PROGRAM P4_01_Write
VAR
	stDBParam 				:ST_AuditTrail;	
	tableColumns			:ARRAY [0..5] OF STRING(50) := ['DateTime', 'User', 'Event', 'Description', 'OldValue', 'NewValue'];	

	fbDBWrite				:FB_PLCDBWriteEvt(sNetId:=CONST.AMS_NETID, tTimeout:=DEFAULT_ADS_TIMEOUT);	
	bWrite					:BOOL;
	

	
	fbRecipeProdValue		:ARRAY[0..9] OF FB_WriteChange;
	fbRecipeProdStrings		:ARRAY[0..9] OF FB_WriteChange_STR;
	fbRecipeProdClick		:ARRAY[0..9] OF FB_WriteClick;
	bRecipeProdChange		:ARRAY[0..19] OF BOOL;
	
	fbRecipeCleanValue		:ARRAY[0..29] OF FB_WriteChange;
	fbRecipeCleanStrings	:ARRAY[0..29] OF FB_WriteChange_STR;
	fbRecipeCleanClick		:ARRAY[0..29] OF FB_WriteClick;
	bRecipeCleanChange		:ARRAY[0..39] OF BOOL;
	
	fbBatchProdValue		:ARRAY[0..9] OF FB_WriteChange;
	fbBatchProdStrings		:ARRAY[0..9] OF FB_WriteChange_STR;
	fbBatchProdClick		:ARRAY[0..9] OF FB_WriteClick;
	bBatchProdChange		:ARRAY[0..19] OF BOOL;
	
	fbBatchCleanValue		:ARRAY[0..29] OF FB_WriteChange;
	fbBatchCleanStrings		:ARRAY[0..29] OF FB_WriteChange_STR;
	fbBatchCleanClick		:ARRAY[0..29] OF FB_WriteClick;
	bBatchCleanChange		:ARRAY[0..39] OF BOOL;
	
	
	fbSettingsChange		:ARRAY[0..19] OF FB_WriteChange;
	bSettingsChange			:ARRAY[0..19] OF BOOL;	
	
	fbAlarmsettChange		:ARRAY[0..9] OF FB_WriteChange;
	bAlarmsettChange		:ARRAY[0..9] OF BOOL;
	
	fbOperatorAction		:ARRAY[0..39] OF FB_WriteClick;
	bOperatorAction			:ARRAY[0..39] OF BOOL;

	bScanBatchParams		:BOOL;
	
END_VAR
VAR // added by the converter: edge detectors and wires of the graphical bodies
    _rt1 : R_TRIG;
END_VAR

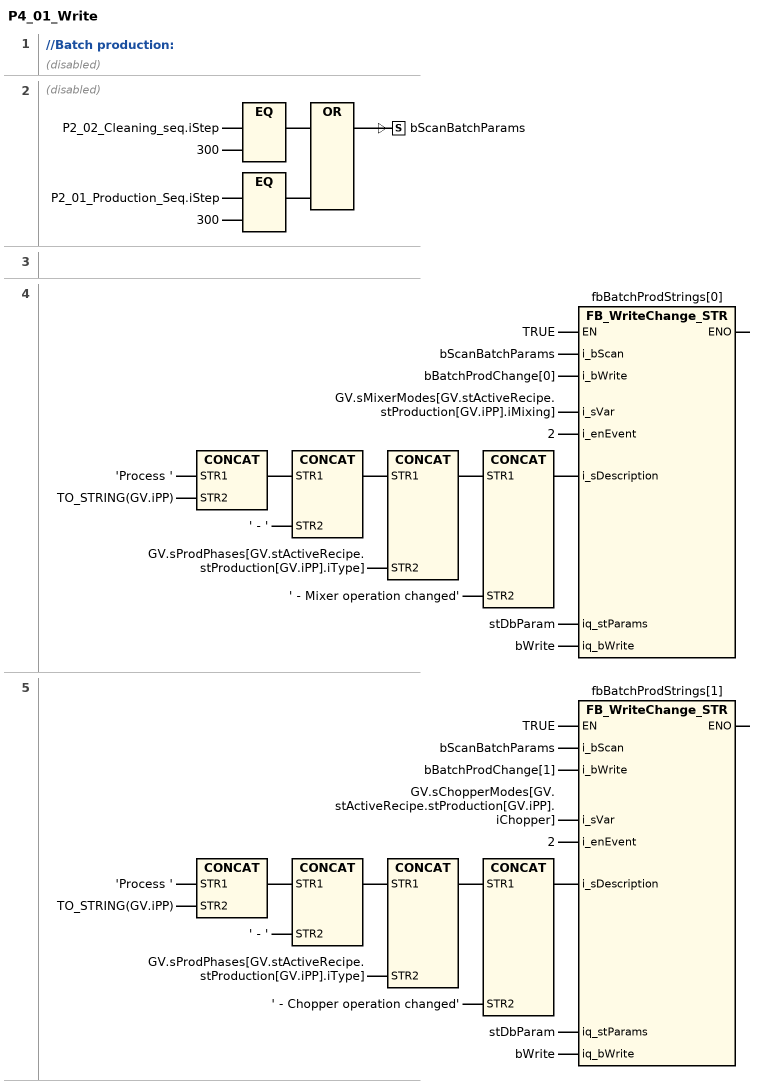
// NETWORK 1 (disabled)
// label: //Batch production

// NETWORK 2 (disabled)
// _rt1(CLK := P2_02_Cleaning_seq.iStep = 300 OR P2_01_Production_Seq.iStep = 300);
// bScanBatchParams S= _rt1.Q;

// NETWORK 3

// NETWORK 4
fbBatchProdStrings[0](
    i_bScan := bScanBatchParams,
    i_bWrite := bBatchProdChange[0],
    i_sVar := GV.sMixerModes[GV.stActiveRecipe.stProduction[GV.iPP].iMixing],
    i_enEvent := 2,
    i_sDescription := CONCAT(STR1 := CONCAT(STR1 := CONCAT(STR1 := CONCAT(STR1 := 'Process ', STR2 := TO_STRING(GV.iPP)), STR2 := ' - '), STR2 := GV.sProdPhases[GV.stActiveRecipe.stProduction[GV.iPP].iType]), STR2 := ' - Mixer operation changed'),
    iq_stParams := stDbParam,
    iq_bWrite := bWrite); // FB_WriteChange_STR

// NETWORK 5
fbBatchProdStrings[1](
    i_bScan := bScanBatchParams,
    i_bWrite := bBatchProdChange[1],
    i_sVar := GV.sChopperModes[GV.stActiveRecipe.stProduction[GV.iPP].iChopper],
    i_enEvent := 2,
    i_sDescription := CONCAT(STR1 := CONCAT(STR1 := CONCAT(STR1 := CONCAT(STR1 := 'Process ', STR2 := TO_STRING(GV.iPP)), STR2 := ' - '), STR2 := GV.sProdPhases[GV.stActiveRecipe.stProduction[GV.iPP].iType]), STR2 := ' - Chopper operation changed'),
    iq_stParams := stDbParam,
    iq_bWrite := bWrite); // FB_WriteChange_STR

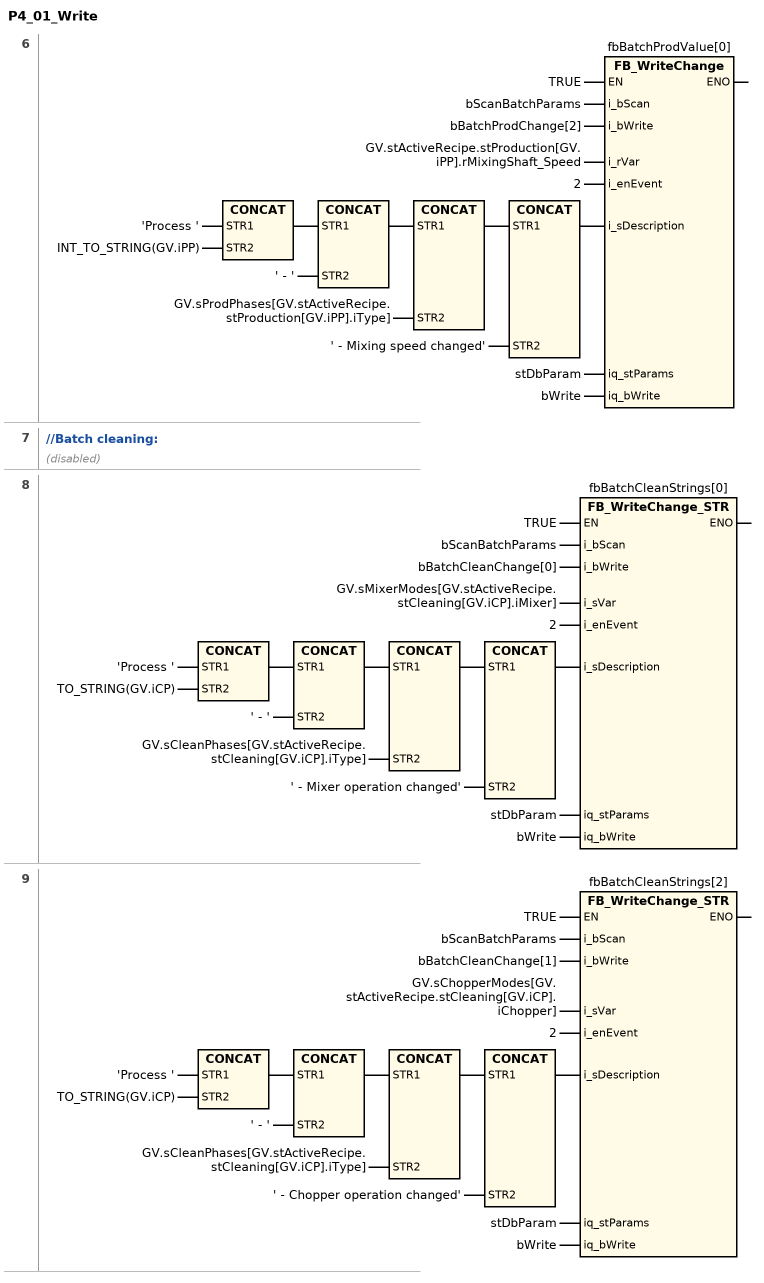
// NETWORK 6
fbBatchProdValue[0](
    i_bScan := bScanBatchParams,
    i_bWrite := bBatchProdChange[2],
    i_rVar := GV.stActiveRecipe.stProduction[GV.iPP].rMixingShaft_Speed,
    i_enEvent := 2,
    i_sDescription := CONCAT(STR1 := CONCAT(STR1 := CONCAT(STR1 := CONCAT(STR1 := 'Process ', STR2 := INT_TO_STRING(GV.iPP)), STR2 := ' - '), STR2 := GV.sProdPhases[GV.stActiveRecipe.stProduction[GV.iPP].iType]), STR2 := ' - Mixing speed changed'),
    iq_stParams := stDbParam,
    iq_bWrite := bWrite); // FB_WriteChange

// NETWORK 7 (disabled)
// label: //Batch cleaning

// NETWORK 8
fbBatchCleanStrings[0](
    i_bScan := bScanBatchParams,
    i_bWrite := bBatchCleanChange[0],
    i_sVar := GV.sMixerModes[GV.stActiveRecipe.stCleaning[GV.iCP].iMixer],
    i_enEvent := 2,
    i_sDescription := CONCAT(STR1 := CONCAT(STR1 := CONCAT(STR1 := CONCAT(STR1 := 'Process ', STR2 := TO_STRING(GV.iCP)), STR2 := ' - '), STR2 := GV.sCleanPhases[GV.stActiveRecipe.stCleaning[GV.iCP].iType]), STR2 := ' - Mixer operation changed'),
    iq_stParams := stDbParam,
    iq_bWrite := bWrite); // FB_WriteChange_STR

// NETWORK 9
fbBatchCleanStrings[2](
    i_bScan := bScanBatchParams,
    i_bWrite := bBatchCleanChange[1],
    i_sVar := GV.sChopperModes[GV.stActiveRecipe.stCleaning[GV.iCP].iChopper],
    i_enEvent := 2,
    i_sDescription := CONCAT(STR1 := CONCAT(STR1 := CONCAT(STR1 := CONCAT(STR1 := 'Process ', STR2 := TO_STRING(GV.iCP)), STR2 := ' - '), STR2 := GV.sCleanPhases[GV.stActiveRecipe.stCleaning[GV.iCP].iType]), STR2 := ' - Chopper operation changed'),
    iq_stParams := stDbParam,
    iq_bWrite := bWrite); // FB_WriteChange_STR

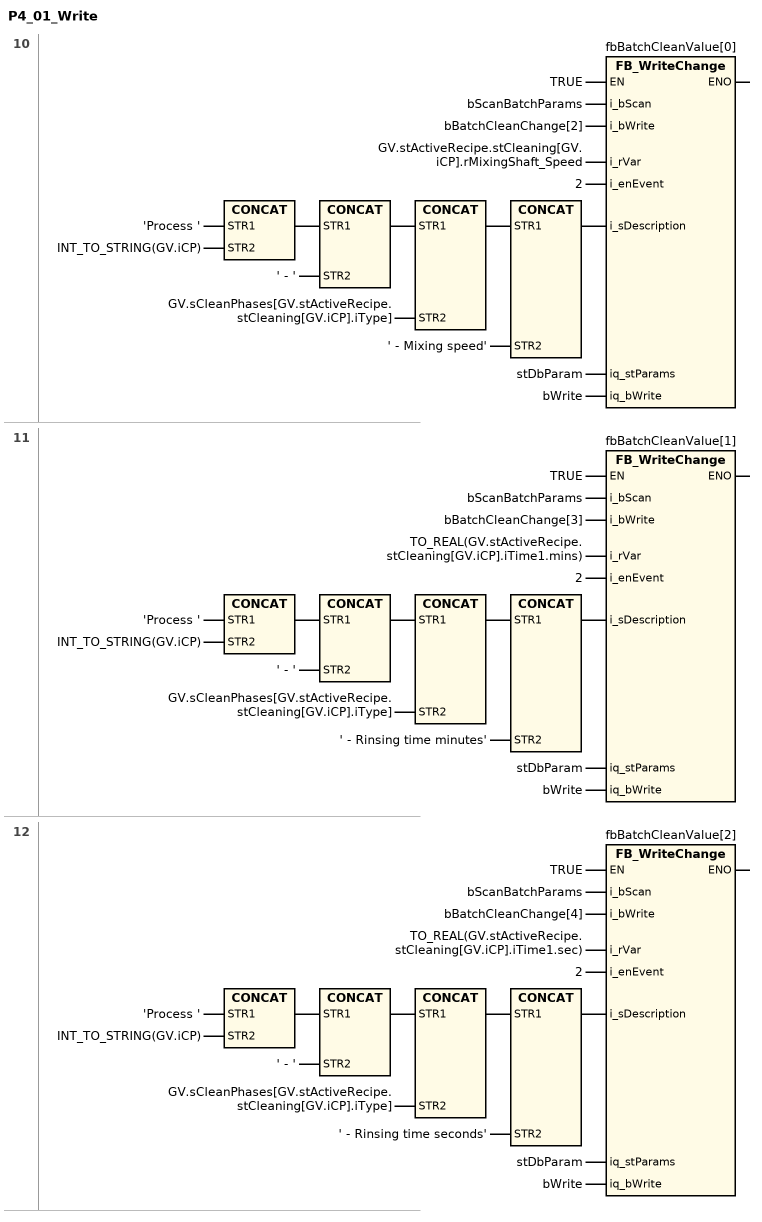
// NETWORK 10
fbBatchCleanValue[0](
    i_bScan := bScanBatchParams,
    i_bWrite := bBatchCleanChange[2],
    i_rVar := GV.stActiveRecipe.stCleaning[GV.iCP].rMixingShaft_Speed,
    i_enEvent := 2,
    i_sDescription := CONCAT(STR1 := CONCAT(STR1 := CONCAT(STR1 := CONCAT(STR1 := 'Process ', STR2 := INT_TO_STRING(GV.iCP)), STR2 := ' - '), STR2 := GV.sCleanPhases[GV.stActiveRecipe.stCleaning[GV.iCP].iType]), STR2 := ' - Mixing speed'),
    iq_stParams := stDbParam,
    iq_bWrite := bWrite); // FB_WriteChange

// NETWORK 11
fbBatchCleanValue[1](
    i_bScan := bScanBatchParams,
    i_bWrite := bBatchCleanChange[3],
    i_rVar := TO_REAL(GV.stActiveRecipe.stCleaning[GV.iCP].iTime1.mins),
    i_enEvent := 2,
    i_sDescription := CONCAT(STR1 := CONCAT(STR1 := CONCAT(STR1 := CONCAT(STR1 := 'Process ', STR2 := INT_TO_STRING(GV.iCP)), STR2 := ' - '), STR2 := GV.sCleanPhases[GV.stActiveRecipe.stCleaning[GV.iCP].iType]), STR2 := ' - Rinsing time minutes'),
    iq_stParams := stDbParam,
    iq_bWrite := bWrite); // FB_WriteChange

// NETWORK 12
fbBatchCleanValue[2](
    i_bScan := bScanBatchParams,
    i_bWrite := bBatchCleanChange[4],
    i_rVar := TO_REAL(GV.stActiveRecipe.stCleaning[GV.iCP].iTime1.sec),
    i_enEvent := 2,
    i_sDescription := CONCAT(STR1 := CONCAT(STR1 := CONCAT(STR1 := CONCAT(STR1 := 'Process ', STR2 := INT_TO_STRING(GV.iCP)), STR2 := ' - '), STR2 := GV.sCleanPhases[GV.stActiveRecipe.stCleaning[GV.iCP].iType]), STR2 := ' - Rinsing time seconds'),
    iq_stParams := stDbParam,
    iq_bWrite := bWrite); // FB_WriteChange

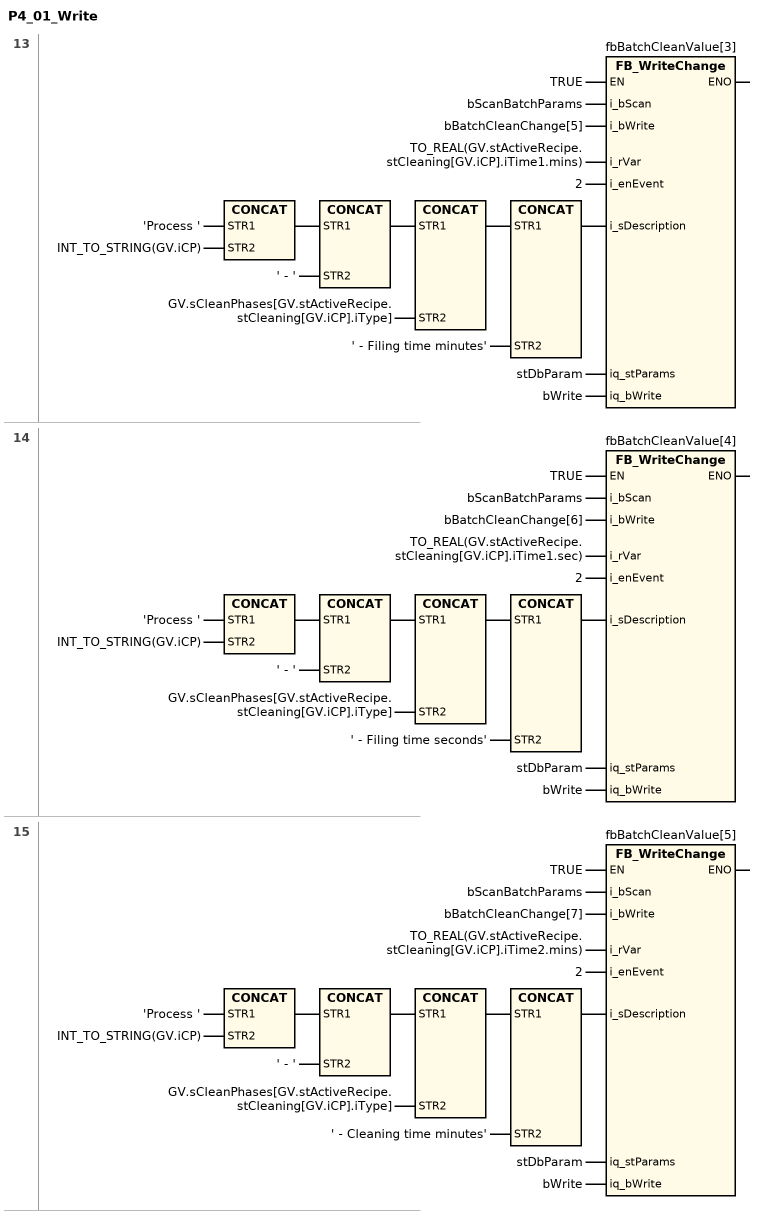
// NETWORK 13
fbBatchCleanValue[3](
    i_bScan := bScanBatchParams,
    i_bWrite := bBatchCleanChange[5],
    i_rVar := TO_REAL(GV.stActiveRecipe.stCleaning[GV.iCP].iTime1.mins),
    i_enEvent := 2,
    i_sDescription := CONCAT(STR1 := CONCAT(STR1 := CONCAT(STR1 := CONCAT(STR1 := 'Process ', STR2 := INT_TO_STRING(GV.iCP)), STR2 := ' - '), STR2 := GV.sCleanPhases[GV.stActiveRecipe.stCleaning[GV.iCP].iType]), STR2 := ' - Filing time minutes'),
    iq_stParams := stDbParam,
    iq_bWrite := bWrite); // FB_WriteChange

// NETWORK 14
fbBatchCleanValue[4](
    i_bScan := bScanBatchParams,
    i_bWrite := bBatchCleanChange[6],
    i_rVar := TO_REAL(GV.stActiveRecipe.stCleaning[GV.iCP].iTime1.sec),
    i_enEvent := 2,
    i_sDescription := CONCAT(STR1 := CONCAT(STR1 := CONCAT(STR1 := CONCAT(STR1 := 'Process ', STR2 := INT_TO_STRING(GV.iCP)), STR2 := ' - '), STR2 := GV.sCleanPhases[GV.stActiveRecipe.stCleaning[GV.iCP].iType]), STR2 := ' - Filing time seconds'),
    iq_stParams := stDbParam,
    iq_bWrite := bWrite); // FB_WriteChange

// NETWORK 15
fbBatchCleanValue[5](
    i_bScan := bScanBatchParams,
    i_bWrite := bBatchCleanChange[7],
    i_rVar := TO_REAL(GV.stActiveRecipe.stCleaning[GV.iCP].iTime2.mins),
    i_enEvent := 2,
    i_sDescription := CONCAT(STR1 := CONCAT(STR1 := CONCAT(STR1 := CONCAT(STR1 := 'Process ', STR2 := INT_TO_STRING(GV.iCP)), STR2 := ' - '), STR2 := GV.sCleanPhases[GV.stActiveRecipe.stCleaning[GV.iCP].iType]), STR2 := ' - Cleaning time minutes'),
    iq_stParams := stDbParam,
    iq_bWrite := bWrite); // FB_WriteChange

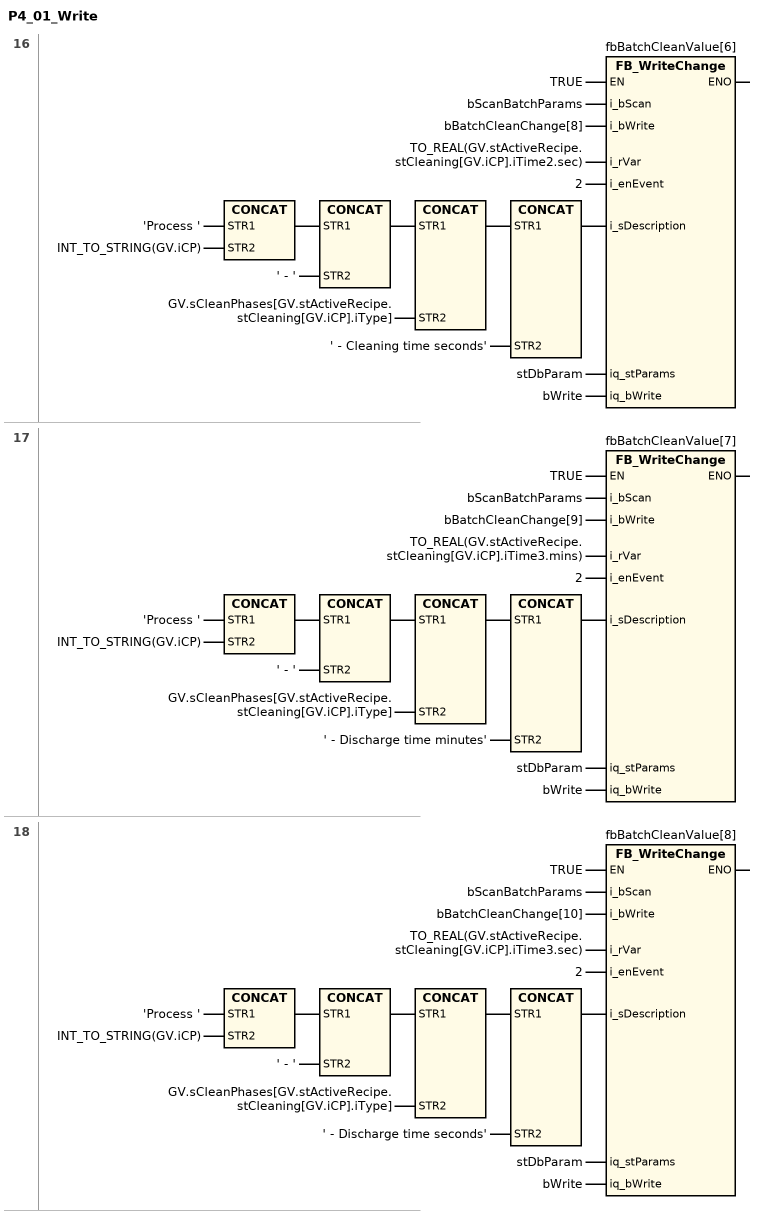
// NETWORK 16
fbBatchCleanValue[6](
    i_bScan := bScanBatchParams,
    i_bWrite := bBatchCleanChange[8],
    i_rVar := TO_REAL(GV.stActiveRecipe.stCleaning[GV.iCP].iTime2.sec),
    i_enEvent := 2,
    i_sDescription := CONCAT(STR1 := CONCAT(STR1 := CONCAT(STR1 := CONCAT(STR1 := 'Process ', STR2 := INT_TO_STRING(GV.iCP)), STR2 := ' - '), STR2 := GV.sCleanPhases[GV.stActiveRecipe.stCleaning[GV.iCP].iType]), STR2 := ' - Cleaning time seconds'),
    iq_stParams := stDbParam,
    iq_bWrite := bWrite); // FB_WriteChange

// NETWORK 17
fbBatchCleanValue[7](
    i_bScan := bScanBatchParams,
    i_bWrite := bBatchCleanChange[9],
    i_rVar := TO_REAL(GV.stActiveRecipe.stCleaning[GV.iCP].iTime3.mins),
    i_enEvent := 2,
    i_sDescription := CONCAT(STR1 := CONCAT(STR1 := CONCAT(STR1 := CONCAT(STR1 := 'Process ', STR2 := INT_TO_STRING(GV.iCP)), STR2 := ' - '), STR2 := GV.sCleanPhases[GV.stActiveRecipe.stCleaning[GV.iCP].iType]), STR2 := ' - Discharge time minutes'),
    iq_stParams := stDbParam,
    iq_bWrite := bWrite); // FB_WriteChange

// NETWORK 18
fbBatchCleanValue[8](
    i_bScan := bScanBatchParams,
    i_bWrite := bBatchCleanChange[10],
    i_rVar := TO_REAL(GV.stActiveRecipe.stCleaning[GV.iCP].iTime3.sec),
    i_enEvent := 2,
    i_sDescription := CONCAT(STR1 := CONCAT(STR1 := CONCAT(STR1 := CONCAT(STR1 := 'Process ', STR2 := INT_TO_STRING(GV.iCP)), STR2 := ' - '), STR2 := GV.sCleanPhases[GV.stActiveRecipe.stCleaning[GV.iCP].iType]), STR2 := ' - Discharge time seconds'),
    iq_stParams := stDbParam,
    iq_bWrite := bWrite); // FB_WriteChange

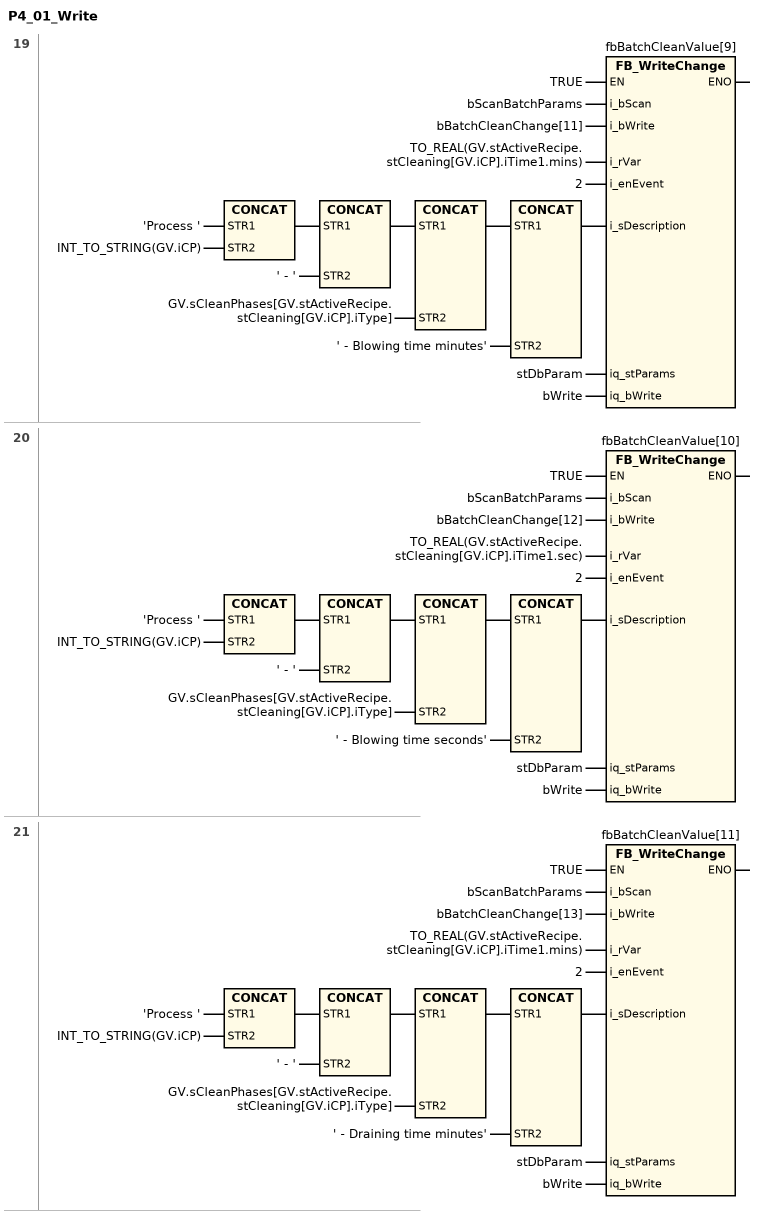
// NETWORK 19
fbBatchCleanValue[9](
    i_bScan := bScanBatchParams,
    i_bWrite := bBatchCleanChange[11],
    i_rVar := TO_REAL(GV.stActiveRecipe.stCleaning[GV.iCP].iTime1.mins),
    i_enEvent := 2,
    i_sDescription := CONCAT(STR1 := CONCAT(STR1 := CONCAT(STR1 := CONCAT(STR1 := 'Process ', STR2 := INT_TO_STRING(GV.iCP)), STR2 := ' - '), STR2 := GV.sCleanPhases[GV.stActiveRecipe.stCleaning[GV.iCP].iType]), STR2 := ' - Blowing time minutes'),
    iq_stParams := stDbParam,
    iq_bWrite := bWrite); // FB_WriteChange

// NETWORK 20
fbBatchCleanValue[10](
    i_bScan := bScanBatchParams,
    i_bWrite := bBatchCleanChange[12],
    i_rVar := TO_REAL(GV.stActiveRecipe.stCleaning[GV.iCP].iTime1.sec),
    i_enEvent := 2,
    i_sDescription := CONCAT(STR1 := CONCAT(STR1 := CONCAT(STR1 := CONCAT(STR1 := 'Process ', STR2 := INT_TO_STRING(GV.iCP)), STR2 := ' - '), STR2 := GV.sCleanPhases[GV.stActiveRecipe.stCleaning[GV.iCP].iType]), STR2 := ' - Blowing time seconds'),
    iq_stParams := stDbParam,
    iq_bWrite := bWrite); // FB_WriteChange

// NETWORK 21
fbBatchCleanValue[11](
    i_bScan := bScanBatchParams,
    i_bWrite := bBatchCleanChange[13],
    i_rVar := TO_REAL(GV.stActiveRecipe.stCleaning[GV.iCP].iTime1.mins),
    i_enEvent := 2,
    i_sDescription := CONCAT(STR1 := CONCAT(STR1 := CONCAT(STR1 := CONCAT(STR1 := 'Process ', STR2 := INT_TO_STRING(GV.iCP)), STR2 := ' - '), STR2 := GV.sCleanPhases[GV.stActiveRecipe.stCleaning[GV.iCP].iType]), STR2 := ' - Draining time minutes'),
    iq_stParams := stDbParam,
    iq_bWrite := bWrite); // FB_WriteChange

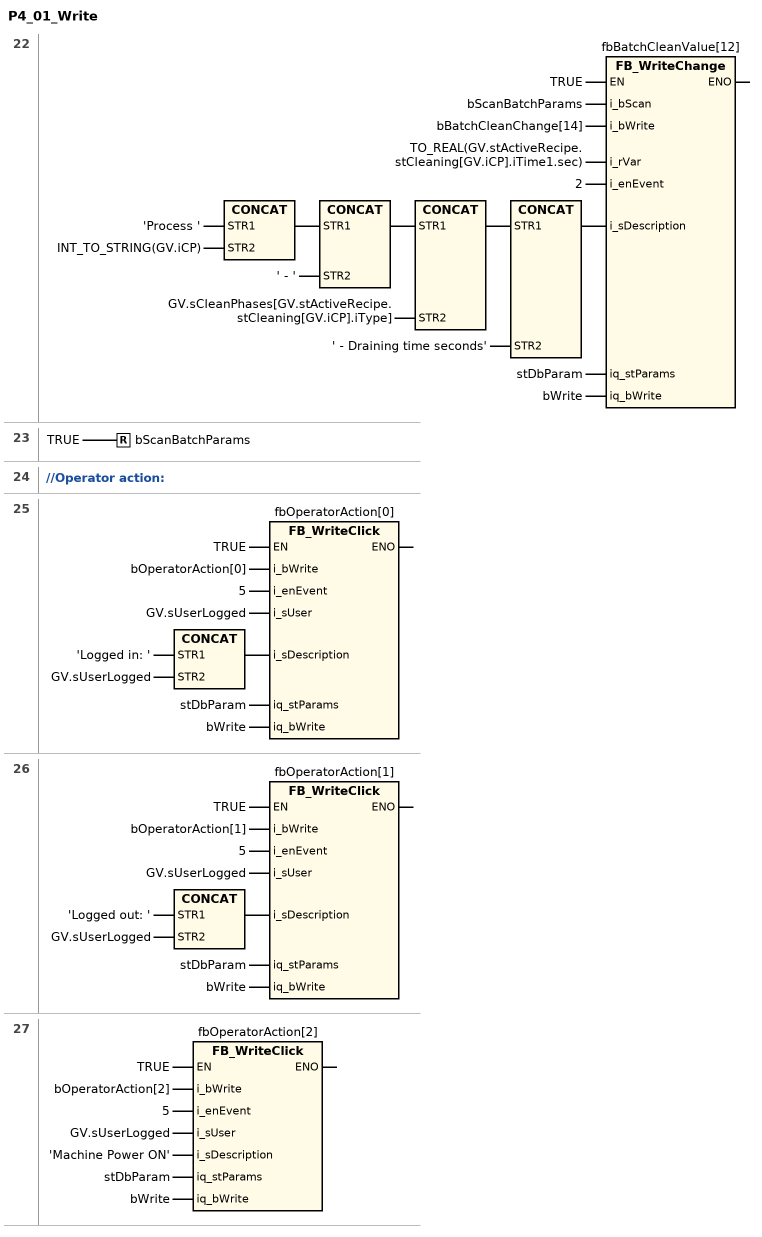
// NETWORK 22
fbBatchCleanValue[12](
    i_bScan := bScanBatchParams,
    i_bWrite := bBatchCleanChange[14],
    i_rVar := TO_REAL(GV.stActiveRecipe.stCleaning[GV.iCP].iTime1.sec),
    i_enEvent := 2,
    i_sDescription := CONCAT(STR1 := CONCAT(STR1 := CONCAT(STR1 := CONCAT(STR1 := 'Process ', STR2 := INT_TO_STRING(GV.iCP)), STR2 := ' - '), STR2 := GV.sCleanPhases[GV.stActiveRecipe.stCleaning[GV.iCP].iType]), STR2 := ' - Draining time seconds'),
    iq_stParams := stDbParam,
    iq_bWrite := bWrite); // FB_WriteChange

// NETWORK 23
bScanBatchParams R= TRUE;

// NETWORK 24
// label: //Operator action

// NETWORK 25
fbOperatorAction[0](
    i_bWrite := bOperatorAction[0],
    i_enEvent := 5,
    i_sUser := GV.sUserLogged,
    i_sDescription := CONCAT(STR1 := 'Logged in: ', STR2 := GV.sUserLogged),
    iq_stParams := stDbParam,
    iq_bWrite := bWrite); // FB_WriteClick

// NETWORK 26
fbOperatorAction[1](
    i_bWrite := bOperatorAction[1],
    i_enEvent := 5,
    i_sUser := GV.sUserLogged,
    i_sDescription := CONCAT(STR1 := 'Logged out: ', STR2 := GV.sUserLogged),
    iq_stParams := stDbParam,
    iq_bWrite := bWrite); // FB_WriteClick

// NETWORK 27
fbOperatorAction[2](
    i_bWrite := bOperatorAction[2],
    i_enEvent := 5,
    i_sUser := GV.sUserLogged,
    i_sDescription := 'Machine Power ON',
    iq_stParams := stDbParam,
    iq_bWrite := bWrite); // FB_WriteClick

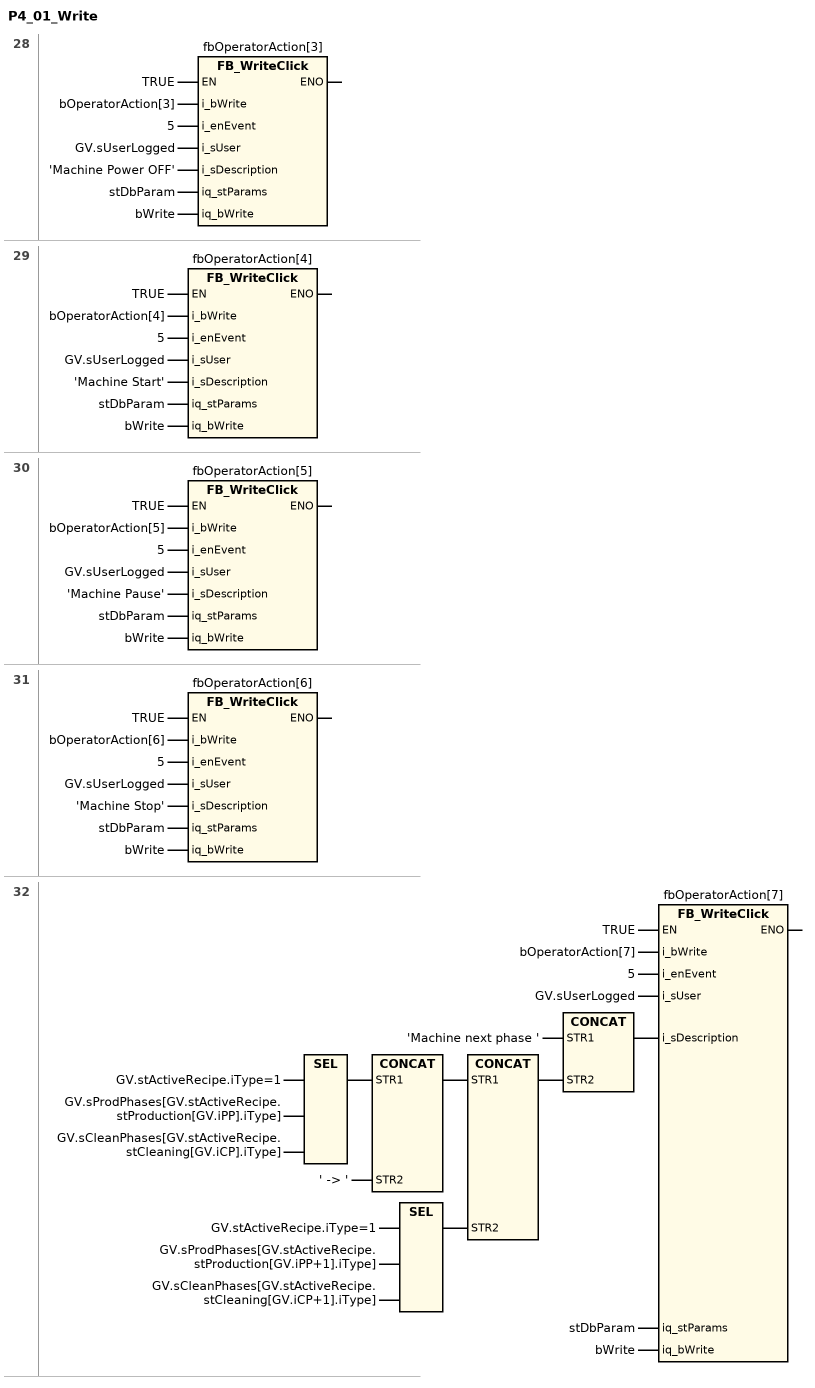
// NETWORK 28
fbOperatorAction[3](
    i_bWrite := bOperatorAction[3],
    i_enEvent := 5,
    i_sUser := GV.sUserLogged,
    i_sDescription := 'Machine Power OFF',
    iq_stParams := stDbParam,
    iq_bWrite := bWrite); // FB_WriteClick

// NETWORK 29
fbOperatorAction[4](
    i_bWrite := bOperatorAction[4],
    i_enEvent := 5,
    i_sUser := GV.sUserLogged,
    i_sDescription := 'Machine Start',
    iq_stParams := stDbParam,
    iq_bWrite := bWrite); // FB_WriteClick

// NETWORK 30
fbOperatorAction[5](
    i_bWrite := bOperatorAction[5],
    i_enEvent := 5,
    i_sUser := GV.sUserLogged,
    i_sDescription := 'Machine Pause',
    iq_stParams := stDbParam,
    iq_bWrite := bWrite); // FB_WriteClick

// NETWORK 31
fbOperatorAction[6](
    i_bWrite := bOperatorAction[6],
    i_enEvent := 5,
    i_sUser := GV.sUserLogged,
    i_sDescription := 'Machine Stop',
    iq_stParams := stDbParam,
    iq_bWrite := bWrite); // FB_WriteClick

// NETWORK 32
fbOperatorAction[7](
    i_bWrite := bOperatorAction[7],
    i_enEvent := 5,
    i_sUser := GV.sUserLogged,
    i_sDescription := CONCAT(STR1 := 'Machine next phase ', STR2 := CONCAT(STR1 := CONCAT(STR1 := SEL(GV.stActiveRecipe.iType=1, GV.sProdPhases[GV.stActiveRecipe.stProduction[GV.iPP].iType], GV.sCleanPhases[GV.stActiveRecipe.stCleaning[GV.iCP].iType]), STR2 := ' -> '), STR2 := SEL(GV.stActiveRecipe.iType=1, GV.sProdPhases[GV.stActiveRecipe.stProduction[GV.iPP+1].iType], GV.sCleanPhases[GV.stActiveRecipe.stCleaning[GV.iCP+1].iType]))),
    iq_stParams := stDbParam,
    iq_bWrite := bWrite); // FB_WriteClick

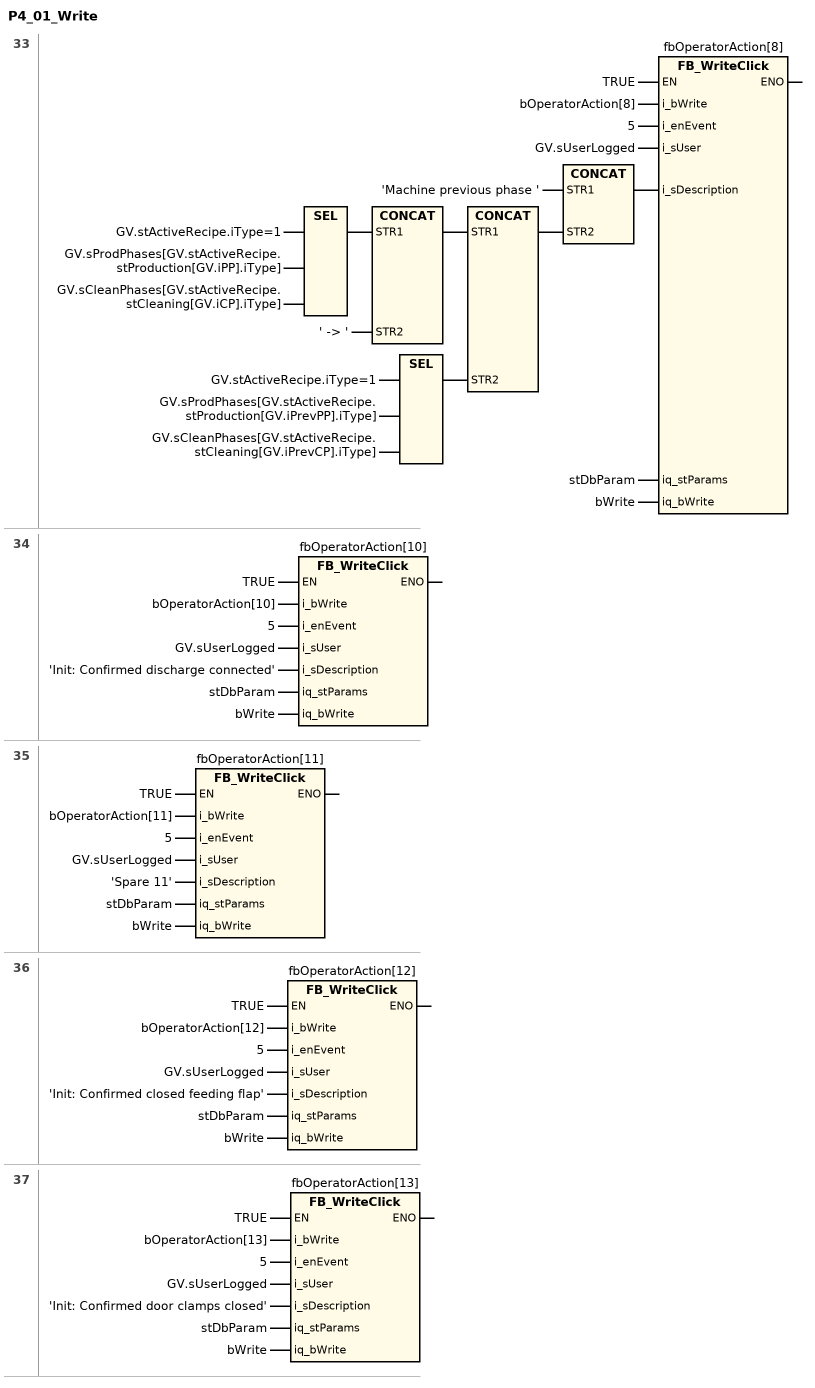
// NETWORK 33
fbOperatorAction[8](
    i_bWrite := bOperatorAction[8],
    i_enEvent := 5,
    i_sUser := GV.sUserLogged,
    i_sDescription := CONCAT(STR1 := 'Machine previous phase ', STR2 := CONCAT(STR1 := CONCAT(STR1 := SEL(GV.stActiveRecipe.iType=1, GV.sProdPhases[GV.stActiveRecipe.stProduction[GV.iPP].iType], GV.sCleanPhases[GV.stActiveRecipe.stCleaning[GV.iCP].iType]), STR2 := ' -> '), STR2 := SEL(GV.stActiveRecipe.iType=1, GV.sProdPhases[GV.stActiveRecipe.stProduction[GV.iPrevPP].iType], GV.sCleanPhases[GV.stActiveRecipe.stCleaning[GV.iPrevCP].iType]))),
    iq_stParams := stDbParam,
    iq_bWrite := bWrite); // FB_WriteClick

// NETWORK 34
fbOperatorAction[10](
    i_bWrite := bOperatorAction[10],
    i_enEvent := 5,
    i_sUser := GV.sUserLogged,
    i_sDescription := 'Init: Confirmed discharge connected',
    iq_stParams := stDbParam,
    iq_bWrite := bWrite); // FB_WriteClick

// NETWORK 35
fbOperatorAction[11](
    i_bWrite := bOperatorAction[11],
    i_enEvent := 5,
    i_sUser := GV.sUserLogged,
    i_sDescription := 'Spare 11',
    iq_stParams := stDbParam,
    iq_bWrite := bWrite); // FB_WriteClick

// NETWORK 36
fbOperatorAction[12](
    i_bWrite := bOperatorAction[12],
    i_enEvent := 5,
    i_sUser := GV.sUserLogged,
    i_sDescription := 'Init: Confirmed closed feeding flap',
    iq_stParams := stDbParam,
    iq_bWrite := bWrite); // FB_WriteClick

// NETWORK 37
fbOperatorAction[13](
    i_bWrite := bOperatorAction[13],
    i_enEvent := 5,
    i_sUser := GV.sUserLogged,
    i_sDescription := 'Init: Confirmed door clamps closed',
    iq_stParams := stDbParam,
    iq_bWrite := bWrite); // FB_WriteClick

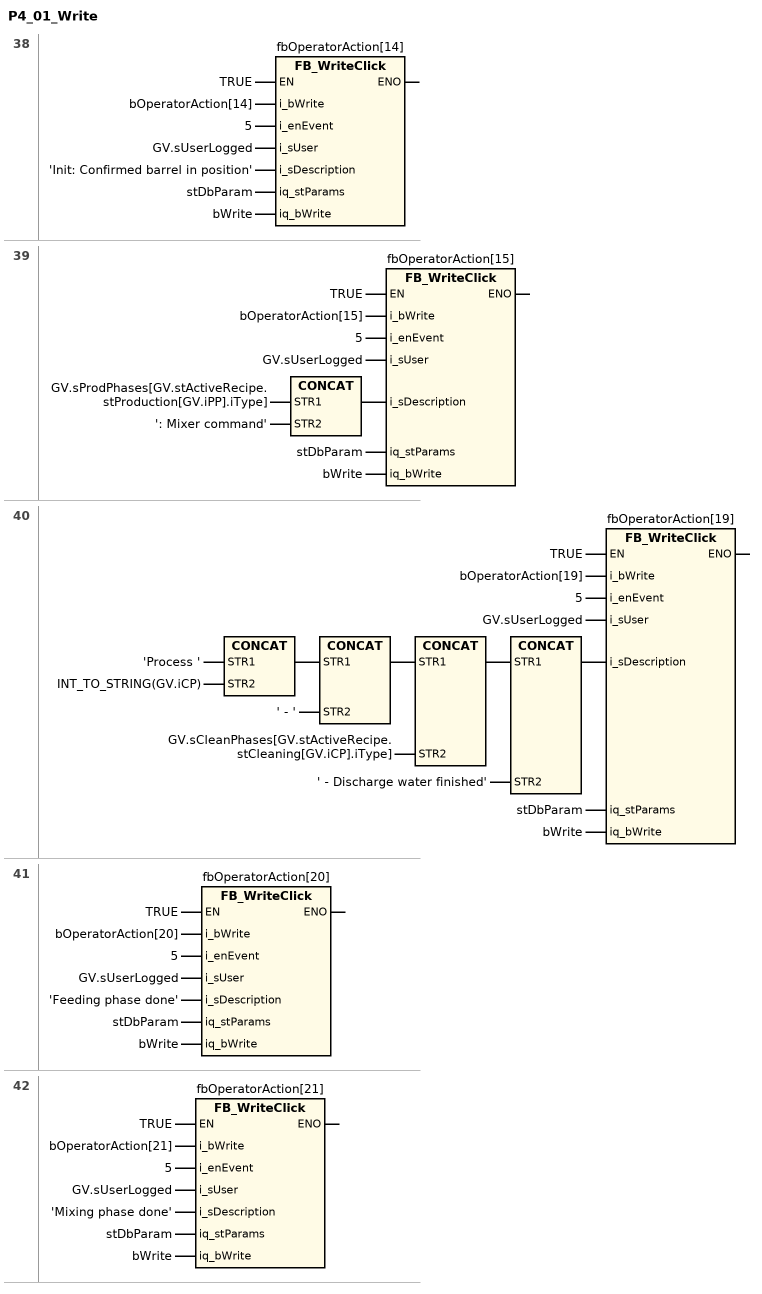
// NETWORK 38
fbOperatorAction[14](
    i_bWrite := bOperatorAction[14],
    i_enEvent := 5,
    i_sUser := GV.sUserLogged,
    i_sDescription := 'Init: Confirmed barrel in position',
    iq_stParams := stDbParam,
    iq_bWrite := bWrite); // FB_WriteClick

// NETWORK 39
fbOperatorAction[15](
    i_bWrite := bOperatorAction[15],
    i_enEvent := 5,
    i_sUser := GV.sUserLogged,
    i_sDescription := CONCAT(STR1 := GV.sProdPhases[GV.stActiveRecipe.stProduction[GV.iPP].iType], STR2 := ': Mixer command'),
    iq_stParams := stDbParam,
    iq_bWrite := bWrite); // FB_WriteClick

// NETWORK 40
fbOperatorAction[19](
    i_bWrite := bOperatorAction[19],
    i_enEvent := 5,
    i_sUser := GV.sUserLogged,
    i_sDescription := CONCAT(STR1 := CONCAT(STR1 := CONCAT(STR1 := CONCAT(STR1 := 'Process ', STR2 := INT_TO_STRING(GV.iCP)), STR2 := ' - '), STR2 := GV.sCleanPhases[GV.stActiveRecipe.stCleaning[GV.iCP].iType]), STR2 := ' - Discharge water finished'),
    iq_stParams := stDbParam,
    iq_bWrite := bWrite); // FB_WriteClick

// NETWORK 41
fbOperatorAction[20](
    i_bWrite := bOperatorAction[20],
    i_enEvent := 5,
    i_sUser := GV.sUserLogged,
    i_sDescription := 'Feeding phase done',
    iq_stParams := stDbParam,
    iq_bWrite := bWrite); // FB_WriteClick

// NETWORK 42
fbOperatorAction[21](
    i_bWrite := bOperatorAction[21],
    i_enEvent := 5,
    i_sUser := GV.sUserLogged,
    i_sDescription := 'Mixing phase done',
    iq_stParams := stDbParam,
    iq_bWrite := bWrite); // FB_WriteClick

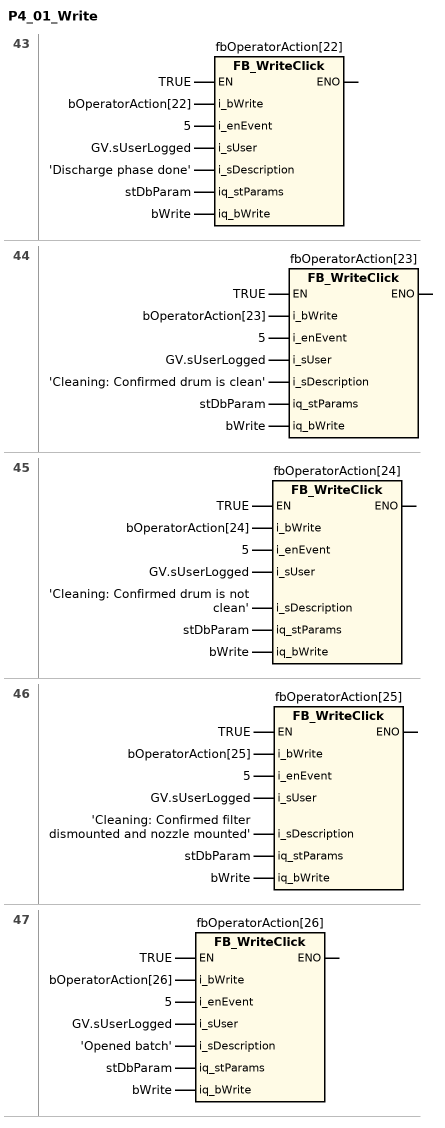
// NETWORK 43
fbOperatorAction[22](
    i_bWrite := bOperatorAction[22],
    i_enEvent := 5,
    i_sUser := GV.sUserLogged,
    i_sDescription := 'Discharge phase done',
    iq_stParams := stDbParam,
    iq_bWrite := bWrite); // FB_WriteClick

// NETWORK 44
fbOperatorAction[23](
    i_bWrite := bOperatorAction[23],
    i_enEvent := 5,
    i_sUser := GV.sUserLogged,
    i_sDescription := 'Cleaning: Confirmed drum is clean',
    iq_stParams := stDbParam,
    iq_bWrite := bWrite); // FB_WriteClick

// NETWORK 45
fbOperatorAction[24](
    i_bWrite := bOperatorAction[24],
    i_enEvent := 5,
    i_sUser := GV.sUserLogged,
    i_sDescription := 'Cleaning: Confirmed drum is not clean',
    iq_stParams := stDbParam,
    iq_bWrite := bWrite); // FB_WriteClick

// NETWORK 46
fbOperatorAction[25](
    i_bWrite := bOperatorAction[25],
    i_enEvent := 5,
    i_sUser := GV.sUserLogged,
    i_sDescription := 'Cleaning: Confirmed filter dismounted and nozzle mounted',
    iq_stParams := stDbParam,
    iq_bWrite := bWrite); // FB_WriteClick

// NETWORK 47
fbOperatorAction[26](
    i_bWrite := bOperatorAction[26],
    i_enEvent := 5,
    i_sUser := GV.sUserLogged,
    i_sDescription := 'Opened batch',
    iq_stParams := stDbParam,
    iq_bWrite := bWrite); // FB_WriteClick

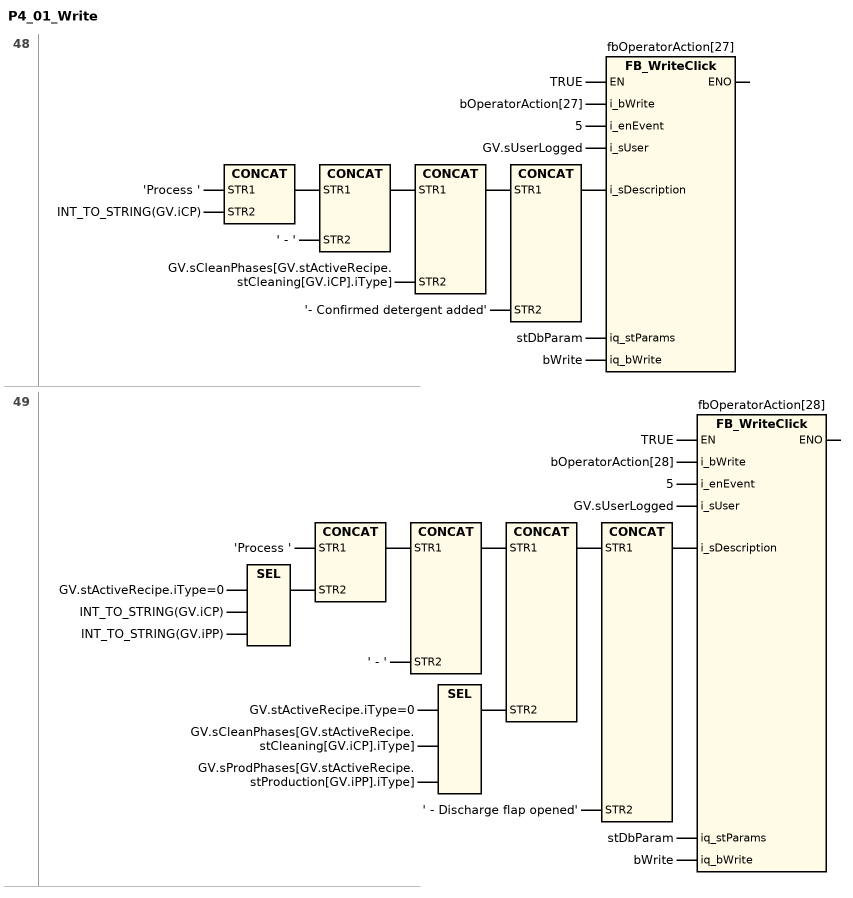
// NETWORK 48
fbOperatorAction[27](
    i_bWrite := bOperatorAction[27],
    i_enEvent := 5,
    i_sUser := GV.sUserLogged,
    i_sDescription := CONCAT(STR1 := CONCAT(STR1 := CONCAT(STR1 := CONCAT(STR1 := 'Process ', STR2 := INT_TO_STRING(GV.iCP)), STR2 := ' - '), STR2 := GV.sCleanPhases[GV.stActiveRecipe.stCleaning[GV.iCP].iType]), STR2 := '- Confirmed detergent added'),
    iq_stParams := stDbParam,
    iq_bWrite := bWrite); // FB_WriteClick

// NETWORK 49
fbOperatorAction[28](
    i_bWrite := bOperatorAction[28],
    i_enEvent := 5,
    i_sUser := GV.sUserLogged,
    i_sDescription := CONCAT(STR1 := CONCAT(STR1 := CONCAT(STR1 := CONCAT(STR1 := 'Process ', STR2 := SEL(GV.stActiveRecipe.iType=0, INT_TO_STRING(GV.iCP), INT_TO_STRING(GV.iPP))), STR2 := ' - '), STR2 := SEL(GV.stActiveRecipe.iType=0, GV.sCleanPhases[GV.stActiveRecipe.stCleaning[GV.iCP].iType], GV.sProdPhases[GV.stActiveRecipe.stProduction[GV.iPP].iType])), STR2 := ' - Discharge flap opened'),
    iq_stParams := stDbParam,
    iq_bWrite := bWrite); // FB_WriteClick

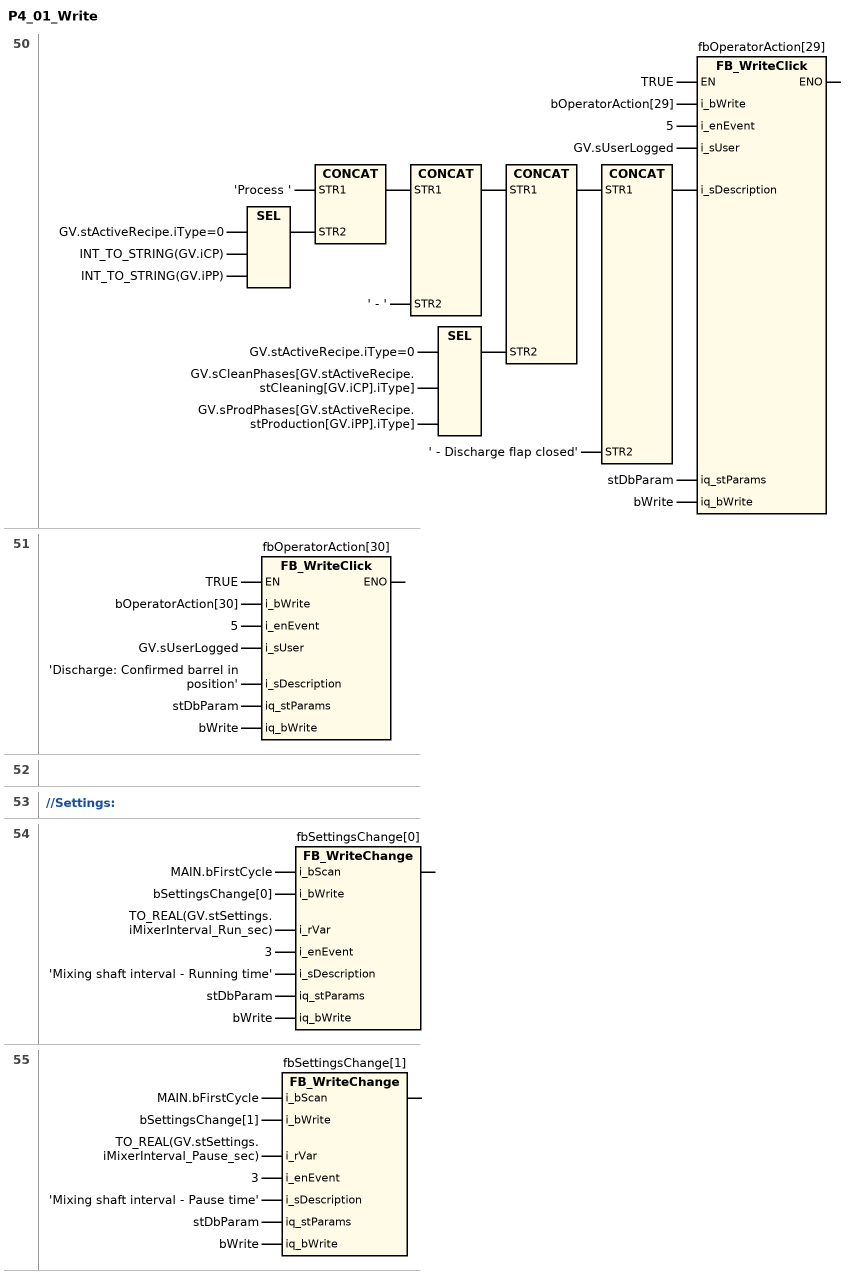
// NETWORK 50
fbOperatorAction[29](
    i_bWrite := bOperatorAction[29],
    i_enEvent := 5,
    i_sUser := GV.sUserLogged,
    i_sDescription := CONCAT(STR1 := CONCAT(STR1 := CONCAT(STR1 := CONCAT(STR1 := 'Process ', STR2 := SEL(GV.stActiveRecipe.iType=0, INT_TO_STRING(GV.iCP), INT_TO_STRING(GV.iPP))), STR2 := ' - '), STR2 := SEL(GV.stActiveRecipe.iType=0, GV.sCleanPhases[GV.stActiveRecipe.stCleaning[GV.iCP].iType], GV.sProdPhases[GV.stActiveRecipe.stProduction[GV.iPP].iType])), STR2 := ' - Discharge flap closed'),
    iq_stParams := stDbParam,
    iq_bWrite := bWrite); // FB_WriteClick

// NETWORK 51
fbOperatorAction[30](
    i_bWrite := bOperatorAction[30],
    i_enEvent := 5,
    i_sUser := GV.sUserLogged,
    i_sDescription := 'Discharge: Confirmed barrel in position',
    iq_stParams := stDbParam,
    iq_bWrite := bWrite); // FB_WriteClick

// NETWORK 52

// NETWORK 53
// label: //Settings

// NETWORK 54
fbSettingsChange[0](
    i_bScan := MAIN.bFirstCycle,
    i_bWrite := bSettingsChange[0],
    i_rVar := TO_REAL(GV.stSettings.iMixerInterval_Run_sec),
    i_enEvent := 3,
    i_sDescription := 'Mixing shaft interval - Running time',
    iq_stParams := stDbParam,
    iq_bWrite := bWrite); // FB_WriteChange

// NETWORK 55
fbSettingsChange[1](
    i_bScan := MAIN.bFirstCycle,
    i_bWrite := bSettingsChange[1],
    i_rVar := TO_REAL(GV.stSettings.iMixerInterval_Pause_sec),
    i_enEvent := 3,
    i_sDescription := 'Mixing shaft interval - Pause time',
    iq_stParams := stDbParam,
    iq_bWrite := bWrite); // FB_WriteChange

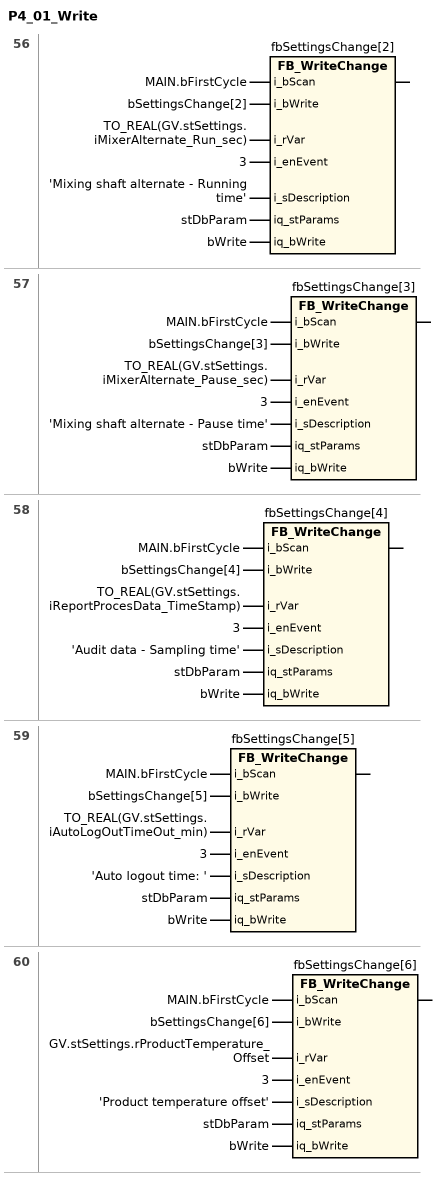
// NETWORK 56
fbSettingsChange[2](
    i_bScan := MAIN.bFirstCycle,
    i_bWrite := bSettingsChange[2],
    i_rVar := TO_REAL(GV.stSettings.iMixerAlternate_Run_sec),
    i_enEvent := 3,
    i_sDescription := 'Mixing shaft alternate - Running time',
    iq_stParams := stDbParam,
    iq_bWrite := bWrite); // FB_WriteChange

// NETWORK 57
fbSettingsChange[3](
    i_bScan := MAIN.bFirstCycle,
    i_bWrite := bSettingsChange[3],
    i_rVar := TO_REAL(GV.stSettings.iMixerAlternate_Pause_sec),
    i_enEvent := 3,
    i_sDescription := 'Mixing shaft alternate - Pause time',
    iq_stParams := stDbParam,
    iq_bWrite := bWrite); // FB_WriteChange

// NETWORK 58
fbSettingsChange[4](
    i_bScan := MAIN.bFirstCycle,
    i_bWrite := bSettingsChange[4],
    i_rVar := TO_REAL(GV.stSettings.iReportProcesData_TimeStamp),
    i_enEvent := 3,
    i_sDescription := 'Audit data - Sampling time',
    iq_stParams := stDbParam,
    iq_bWrite := bWrite); // FB_WriteChange

// NETWORK 59
fbSettingsChange[5](
    i_bScan := MAIN.bFirstCycle,
    i_bWrite := bSettingsChange[5],
    i_rVar := TO_REAL(GV.stSettings.iAutoLogOutTimeOut_min),
    i_enEvent := 3,
    i_sDescription := 'Auto logout time: ',
    iq_stParams := stDbParam,
    iq_bWrite := bWrite); // FB_WriteChange

// NETWORK 60
fbSettingsChange[6](
    i_bScan := MAIN.bFirstCycle,
    i_bWrite := bSettingsChange[6],
    i_rVar := GV.stSettings.rProductTemperature_Offset,
    i_enEvent := 3,
    i_sDescription := 'Product temperature offset',
    iq_stParams := stDbParam,
    iq_bWrite := bWrite); // FB_WriteChange

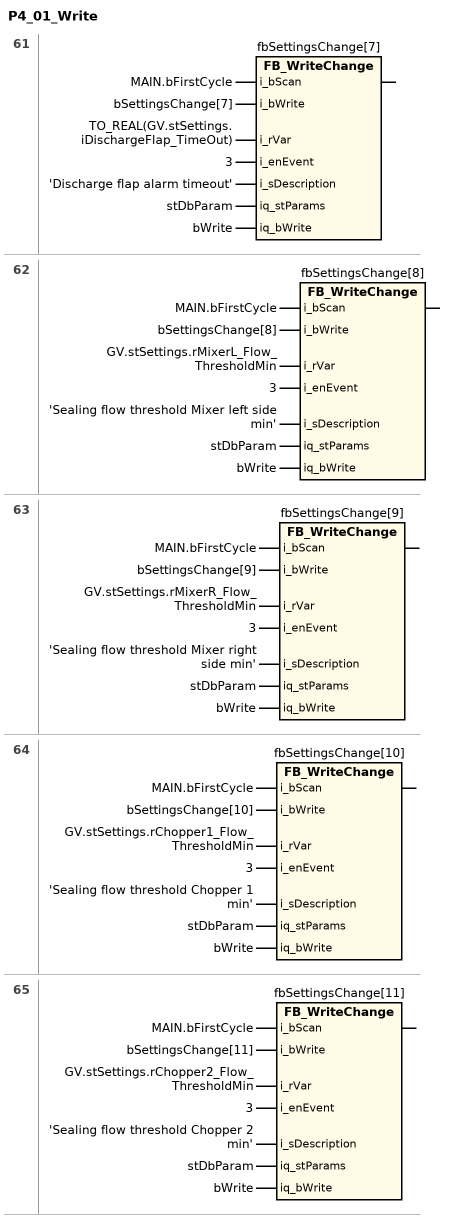
// NETWORK 61
fbSettingsChange[7](
    i_bScan := MAIN.bFirstCycle,
    i_bWrite := bSettingsChange[7],
    i_rVar := TO_REAL(GV.stSettings.iDischargeFlap_TimeOut),
    i_enEvent := 3,
    i_sDescription := 'Discharge flap alarm timeout',
    iq_stParams := stDbParam,
    iq_bWrite := bWrite); // FB_WriteChange

// NETWORK 62
fbSettingsChange[8](
    i_bScan := MAIN.bFirstCycle,
    i_bWrite := bSettingsChange[8],
    i_rVar := GV.stSettings.rMixerL_Flow_ThresholdMin,
    i_enEvent := 3,
    i_sDescription := 'Sealing flow threshold Mixer left side min',
    iq_stParams := stDbParam,
    iq_bWrite := bWrite); // FB_WriteChange

// NETWORK 63
fbSettingsChange[9](
    i_bScan := MAIN.bFirstCycle,
    i_bWrite := bSettingsChange[9],
    i_rVar := GV.stSettings.rMixerR_Flow_ThresholdMin,
    i_enEvent := 3,
    i_sDescription := 'Sealing flow threshold Mixer right side min',
    iq_stParams := stDbParam,
    iq_bWrite := bWrite); // FB_WriteChange

// NETWORK 64
fbSettingsChange[10](
    i_bScan := MAIN.bFirstCycle,
    i_bWrite := bSettingsChange[10],
    i_rVar := GV.stSettings.rChopper1_Flow_ThresholdMin,
    i_enEvent := 3,
    i_sDescription := 'Sealing flow threshold Chopper 1 min',
    iq_stParams := stDbParam,
    iq_bWrite := bWrite); // FB_WriteChange

// NETWORK 65
fbSettingsChange[11](
    i_bScan := MAIN.bFirstCycle,
    i_bWrite := bSettingsChange[11],
    i_rVar := GV.stSettings.rChopper2_Flow_ThresholdMin,
    i_enEvent := 3,
    i_sDescription := 'Sealing flow threshold Chopper 2 min',
    iq_stParams := stDbParam,
    iq_bWrite := bWrite); // FB_WriteChange

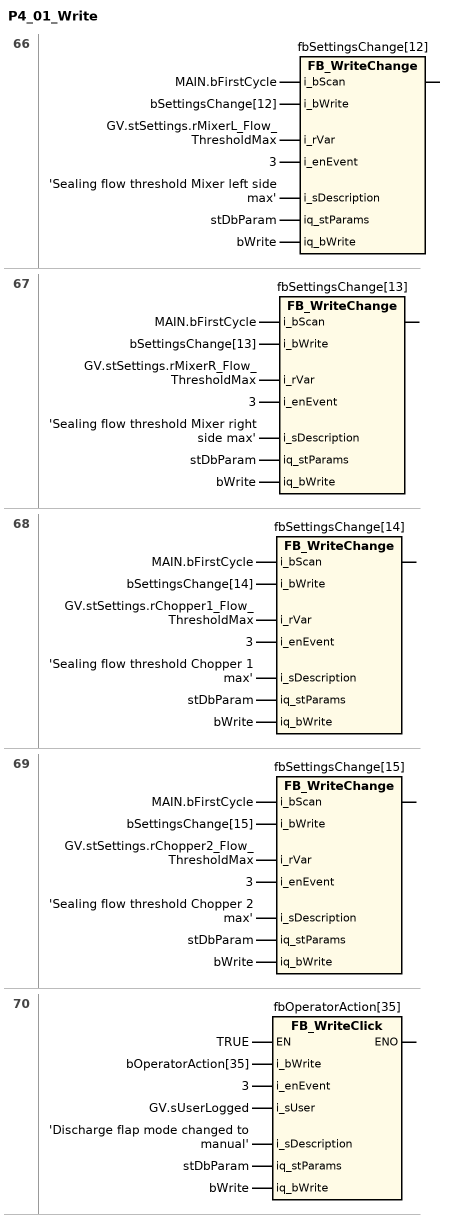
// NETWORK 66
fbSettingsChange[12](
    i_bScan := MAIN.bFirstCycle,
    i_bWrite := bSettingsChange[12],
    i_rVar := GV.stSettings.rMixerL_Flow_ThresholdMax,
    i_enEvent := 3,
    i_sDescription := 'Sealing flow threshold Mixer left side max',
    iq_stParams := stDbParam,
    iq_bWrite := bWrite); // FB_WriteChange

// NETWORK 67
fbSettingsChange[13](
    i_bScan := MAIN.bFirstCycle,
    i_bWrite := bSettingsChange[13],
    i_rVar := GV.stSettings.rMixerR_Flow_ThresholdMax,
    i_enEvent := 3,
    i_sDescription := 'Sealing flow threshold Mixer right side max',
    iq_stParams := stDbParam,
    iq_bWrite := bWrite); // FB_WriteChange

// NETWORK 68
fbSettingsChange[14](
    i_bScan := MAIN.bFirstCycle,
    i_bWrite := bSettingsChange[14],
    i_rVar := GV.stSettings.rChopper1_Flow_ThresholdMax,
    i_enEvent := 3,
    i_sDescription := 'Sealing flow threshold Chopper 1 max',
    iq_stParams := stDbParam,
    iq_bWrite := bWrite); // FB_WriteChange

// NETWORK 69
fbSettingsChange[15](
    i_bScan := MAIN.bFirstCycle,
    i_bWrite := bSettingsChange[15],
    i_rVar := GV.stSettings.rChopper2_Flow_ThresholdMax,
    i_enEvent := 3,
    i_sDescription := 'Sealing flow threshold Chopper 2 max',
    iq_stParams := stDbParam,
    iq_bWrite := bWrite); // FB_WriteChange

// NETWORK 70
fbOperatorAction[35](
    i_bWrite := bOperatorAction[35],
    i_enEvent := 3,
    i_sUser := GV.sUserLogged,
    i_sDescription := 'Discharge flap mode changed to manual',
    iq_stParams := stDbParam,
    iq_bWrite := bWrite); // FB_WriteClick

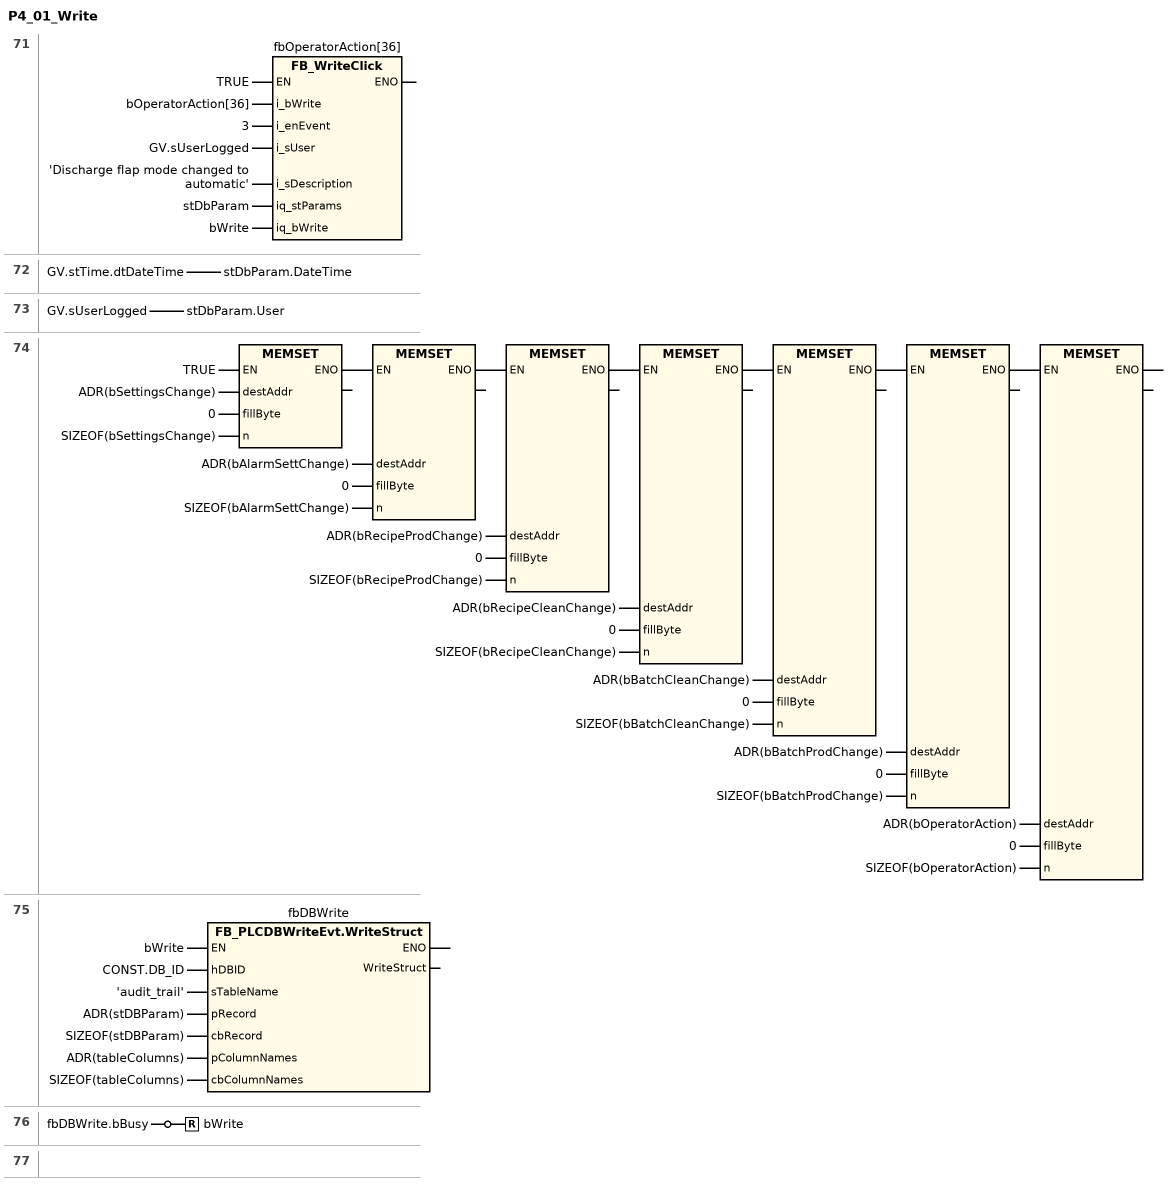
// NETWORK 71
fbOperatorAction[36](
    i_bWrite := bOperatorAction[36],
    i_enEvent := 3,
    i_sUser := GV.sUserLogged,
    i_sDescription := 'Discharge flap mode changed to automatic',
    iq_stParams := stDbParam,
    iq_bWrite := bWrite); // FB_WriteClick

// NETWORK 72
stDbParam.DateTime := GV.stTime.dtDateTime;

// NETWORK 73
stDbParam.User := GV.sUserLogged;

// NETWORK 74
MEMSET(destAddr := ADR(bSettingsChange), fillByte := 0, n := SIZEOF(bSettingsChange));
MEMSET(destAddr := ADR(bAlarmSettChange), fillByte := 0, n := SIZEOF(bAlarmSettChange));
MEMSET(destAddr := ADR(bRecipeProdChange), fillByte := 0, n := SIZEOF(bRecipeProdChange));
MEMSET(destAddr := ADR(bRecipeCleanChange), fillByte := 0, n := SIZEOF(bRecipeCleanChange));
MEMSET(destAddr := ADR(bBatchCleanChange), fillByte := 0, n := SIZEOF(bBatchCleanChange));
MEMSET(destAddr := ADR(bBatchProdChange), fillByte := 0, n := SIZEOF(bBatchProdChange));
MEMSET(destAddr := ADR(bOperatorAction), fillByte := 0, n := SIZEOF(bOperatorAction));

// NETWORK 75
IF bWrite THEN
    fbDBWrite.WriteStruct(
        hDBID := CONST.DB_ID,
        sTableName := 'audit_trail',
        pRecord := ADR(stDBParam),
        cbRecord := SIZEOF(stDBParam),
        pColumnNames := ADR(tableColumns),
        cbColumnNames := SIZEOF(tableColumns));
END_IF

// NETWORK 76
bWrite R= NOT fbDBWrite.bBusy;

// NETWORK 77

END_PROGRAM

(* stored: Version 1.1.0.1
   POU P4_01_Write: Id {a731bf3e-578e-46fd-a95c-8fb35538aecf}, SpecialFunc None *)
